# B&R Automation Studio project test
Automation Studio 4.9

## Configuration Config2

CPU X20CP3685, AutomationRuntime J4.93, Build 6.3.0, Vc V4.73.5

### Hardware
```
X20CP3685 : X20CP3685 v1.9.0.0
  Simulation = 1
  FileDevice1
  FileDeviceName1 = USER
  FileDevicePath1 = USER_PATH
```

## Logical view

Binary libraries used (declarations not repeated): operator, runtime, astime, AsIecCon, ArEventLog, FileIO, MyReadCfg, AsBrStr, sys_lib, standard, brsystem


### Program Logical/readcfg (IEC)

#### Variables.var
```iecst
VAR
	cfgDevice : STRING[32] := 'USER'; (*FileIO device pointing to the USER partition*)
	gMachineCfg : MachineConfiguration_typ;
	cfgFileName : STRING[80] := 'settings.ini';
	cfgIdent : UDINT;
END_VAR
```

#### Main.st
```iecst
PROGRAM _INIT
	cfgIdent := MRC_Open(ADR(cfgDevice), ADR(cfgFileName));

	(* read STRING *)
	MRC_ReadSTRING( cfgIdent, ADR('app_name'), ADR(gMachineCfg.app_name), SIZEOF(gMachineCfg.app_name), ADR('<unknown>') );
	MRC_ReadSTRING( cfgIdent, ADR('database_host'), ADR(gMachineCfg.database_host), SIZEOF(gMachineCfg.database_host), ADR('0.0.0.0') );
	MRC_ReadSTRING( cfgIdent, ADR('log_file_path'), ADR(gMachineCfg.log_file_path), SIZEOF(gMachineCfg.log_file_path), ADR('\') );

	(* read DINT *)
	gMachineCfg.max_connections := MRC_ReadDINT(cfgIdent, ADR('max_connections'), 0);
	gMachineCfg.port_number := MRC_ReadDINT(cfgIdent, ADR('port_number'), 0);
	gMachineCfg.timeout_seconds := MRC_ReadDINT(cfgIdent, ADR('timeout_seconds'), 0);

	(* read BOOL *)
	gMachineCfg.debug_mode := MRC_ReadBOOL(cfgIdent, ADR('debug_mode'), FALSE);
	gMachineCfg.enable_logging := MRC_ReadBOOL(cfgIdent, ADR('enable_logging'), FALSE);
	gMachineCfg.ssl_enabled := MRC_ReadBOOL(cfgIdent, ADR('ssl_enabled'), FALSE);

	(* read LREAL *)
	gMachineCfg.cpu_threshold := MRC_ReadLREAL(cfgIdent, ADR('cpu_threshold'), 0.0);
	gMachineCfg.memory_limit_gb := MRC_ReadLREAL(cfgIdent, ADR('memory_limit_gb'), 0.0);

	MRC_Close(cfgIdent);
	cfgIdent := 0;

	ST_tmp_suspend(0);
END_PROGRAM

PROGRAM _CYCLIC

END_PROGRAM

PROGRAM _EXIT
	IF cfgIdent <> 0 THEN
		MRC_Close(cfgIdent);
		cfgIdent := 0;
	END_IF
END_PROGRAM
```

Listed in the project but not available here: Logical/Global.typ, Logical/Global.var
